// TwinCAT 3 PLC project PlcIotHttpSamplesAwsIotCore
// ProgramVersion: 3.1.4023.0
// libraries:
//   Tc2_Standard, * (Beckhoff Automation GmbH)
//   Tc2_System, * (Beckhoff Automation GmbH)
//   Tc2_Utilities, * (Beckhoff Automation GmbH)
//   Tc3_IotBase, * (Beckhoff Automation GmbH)
//   Tc3_JsonXml, * (Beckhoff Automation GmbH)
//   Tc3_Module, * (Beckhoff Automation GmbH)
// project tree:
//   / PlcTask.TcTTO
//   POUs/AWS IoT Core/ FB_TestHTTP_Get_awsIotShadow.TcPOU, FB_TestHTTP_Post_awsIot.TcPOU
//   POUs/ MAIN.TcPOU
// (motion and I/O tree: see PLC project plciothttpsamplespostman)
// real-time tasks:
//   TASK PlcTask: cycle T#10ms, priority 20, ADS port 350
//   TASK PlcTask1: cycle T#10ms, priority 21, ADS port 351
//   TASK PlcTask2: cycle T#10ms, priority 22, ADS port 352
//   TASK PlcTask3: cycle T#10ms, priority 23, ADS port 353
//   TASK PlcTask4: cycle T#10ms, priority 24, ADS port 354
//   TASK PlcTask5: cycle T#10ms, priority 25, ADS port 355
//   TASK PlcTask6: cycle T#10ms, priority 26, ADS port 356

CONFIGURATION PlcIotHttpSamplesAwsIotCore
    RESOURCE PLC ON TwinCAT3
        TASK PlcTask(INTERVAL := T#10ms, PRIORITY := 22);
    END_RESOURCE
END_CONFIGURATION

// ---- POUs/AWS IoT Core/FB_TestHTTP_Get_awsIotShadow.TcPOU
FUNCTION_BLOCK FB_TestHTTP_Get_awsIotShadow
VAR_INPUT
	bSend				: BOOL;
END_VAR
VAR_IN_OUT
	fbClient			: FB_IotHttpClient;
END_VAR	
VAR_OUTPUT
	bBusy				: BOOL;
	bError				: BOOL;
END_VAR
VAR	
	fbRequest			: FB_IotHttpRequest;
	fbJson				: FB_JsonDomParser;
	nState				: UDINT;
	RisingEdge			: R_TRIG;
	
	bGetContentResult	: BOOL;
	sContent			: STRING(511);
	
	bGetJsonResult		: BOOL;
	jsonDoc				: SJsonValue;
	jsonVal				: SJsonValue;
	sResultValue		: STRING;
	
	nReqCount			: UDINT;
	nResCount			: UDINT;
	nValidResCount		: UDINT;
	nErrCount			: UDINT;	
END_VAR

RisingEdge(CLK:= bSend);
CASE nState OF
0:		
	IF RisingEdge.Q THEN
		IF fbRequest.SendRequest(sUri:='/things/thingName/shadow', fbClient:= fbClient, eRequestType:= ETcIotHttpRequestType.HTTP_GET, 0, 0, 0) THEN				
			nState:= 1;
			nReqCount:= nReqCount+1;
			bBusy:= TRUE;
			bError:= FALSE;
		END_IF					
	END_IF
1:
	IF NOT fbRequest.bBusy THEN
		bError:= TRUE;
		IF NOT fbRequest.bError THEN				 				
			bGetContentResult:= fbRequest.GetContent(pContent:= ADR(sContent), nContentSize:= SIZEOF(sContent), bSetNullTermination:= TRUE);	
			IF fbRequest.nStatusCode >= 200 AND fbRequest.nStatusCode < 300 THEN
				bGetJsonResult:= FALSE;
				jsonDoc:= fbRequest.GetJsonDomContent(fbJson);				
				IF jsonDoc <> 0 THEN
					; // do something with the shadow document
					nValidResCount:= nValidResCount+1;
					bError:= FALSE;
				END_IF
				nResCount:= nResCount+1;					
			END_IF				
		END_IF
		nState:= 0;
		bBusy:= FALSE;
		IF bError THEN
			nErrCount:= nErrCount+1;
		END_IF		
	END_IF  	
END_CASE

END_FUNCTION_BLOCK

// ---- POUs/AWS IoT Core/FB_TestHTTP_Post_awsIot.TcPOU
FUNCTION_BLOCK FB_TestHTTP_Post_awsIot
VAR_INPUT
	bSend				: BOOL;
END_VAR
VAR_IN_OUT
	fbClient			: FB_IotHttpClient;
END_VAR
VAR_OUTPUT
	bBusy				: BOOL;
	bError				: BOOL;
END_VAR

VAR	
	fbRequest			: FB_IotHttpRequest;
	fbJson				: FB_JsonDomParser;
	fbPayload   		: FB_JsonSaxWriter;
	nState				: UDINT;
	RisingEdge			: R_TRIG;
	
	bGetContentResult	: BOOL;
	sContent			: STRING(511);
	
	bGetJsonResult		: BOOL;
	jsonDoc				: SJsonValue;
	jsonVal				: SJsonValue;
	sResultValue		: STRING;
	
	nReqCount			: UDINT;
	nResCount			: UDINT;
	nValidResCount		: UDINT;
	nErrCount			: UDINT;	
END_VAR

RisingEdge(CLK:= bSend);
CASE nState OF
0:		
	IF RisingEdge.Q THEN
		fbPayload.StartObject();
		fbPayload.AddKey('message');
		fbPayload.AddReal(42.42);
		fbPayload.EndObject();
		sContent:= fbPayload.GetDocument();
		fbPayload.ResetDocument();
		IF fbRequest.SendRequest(sUri:='/topics/mytopic?qos=1', fbClient:= fbClient, eRequestType:= ETcIotHttpRequestType.HTTP_POST, pContent:= ADR(sContent), nContentSize:= LEN2(ADR(sContent)), 0) THEN				
			nState:= 1;
			nReqCount:= nReqCount+1;
			bBusy:= TRUE;
			bError:= FALSE;
		END_IF					
	END_IF
1:
	IF NOT fbRequest.bBusy THEN
		bError:= TRUE;
		IF NOT fbRequest.bError THEN				 				
			bGetContentResult:= fbRequest.GetContent(pContent:=ADR(sContent), nContentSize:=SIZEOF(sContent), bSetNullTermination:=TRUE);	
			IF fbRequest.nStatusCode >= 200 AND fbRequest.nStatusCode < 300 THEN
				bGetJsonResult:= FALSE;
				jsonDoc:= fbRequest.GetJsonDomContent(fbJson);				
				IF jsonDoc <> 0 THEN
					bGetJsonResult:= TRUE;
					IF fbJson.HasMember(jsonDoc, 'message')  THEN
						jsonVal:= fbJson.FindMember(jsonDoc, 'message');
						sResultValue:= fbJson.GetString(jsonVal);
						IF sResultValue = 'OK' THEN
							nValidResCount:= nValidResCount+1;
							bError:= FALSE;
						END_IF
					END_IF		
				END_IF
				nResCount:= nResCount+1;					
			END_IF				
		END_IF
		nState:= 0;
		bBusy:= FALSE;
		IF bError THEN
			nErrCount:= nErrCount+1;
		END_IF		
	END_IF  	
END_CASE

END_FUNCTION_BLOCK

// ---- POUs/MAIN.TcPOU
PROGRAM MAIN
VAR
	// trigger command execution for AWS IoT Core samples
	bGetAwsIotShadow, bPostAwsIot 	: BOOL;

	fbHttpClientAwsIot				: FB_IotHttpClient :=(sHostName:='youradress.amazonaws.com',
								  	bKeepAlive:=FALSE, tConnectionTimeout:=T#10S);
								
	fbHttpGetAwsIotShadow			: FB_TestHTTP_Get_awsIotShadow;	
	fbHttpPostAwsIot				: FB_TestHTTP_Post_awsIot;
END_VAR

// init client parameters at startup
IF NOT fbHttpClientAwsIot.bConfigured THEN 
	fbHttpClientAwsIot.stTLS.sCA:= 'C:\TwinCAT\3.1\Config\Certificates\AWS\AmazonRootCA1.pem';
	fbHttpClientAwsIot.stTLS.sCert:= 'C:\TwinCAT\3.1\Config\Certificates\AWS\12345678-certificate.pem.crt';
	fbHttpClientAwsIot.stTLS.sKeyFile:= 'C:\TwinCAT\3.1\Config\Certificates\AWS\12345678-private.pem.key';
	fbHttpClientAwsIot.nHostPort:= 8443;
END_IF

IF fbHttpClientAwsIot.bConfigured THEN
	fbHttpGetAwsIotShadow(bSend:=bGetAwsIotShadow, fbClient:=fbHttpClientAwsIot);
	fbHttpPostAwsIot(bSend:=bPostAwsIot, fbClient:=fbHttpClientAwsIot);
END_IF

fbHttpClientAwsIot.Execute();

END_PROGRAM
